# B&R Automation Studio project UdpReceiverSender
Automation Studio 4.5.3.86 SP

## Configuration Config1

CPU X20CP1585, AutomationRuntime A4.53, Build 4.1.2, Vc V4.52.0

### Task classes (Cpu.sw)
```
Cyclic#4:
  UDP <- UDP.prg
Libraries: AsUDP, runtime
```

### Hardware
```
X20CP1585 : X20CP1585 v1.6.0.0
  Connector IF2:
    ActivateDevice = 1
    Mode = Manual
    InternetAddress = 192.168.32.19
    SubnetMask = 255.255.255.0
  ConfigurationID = UdpReceiverSender_Config1
```

## Logical view

Binary libraries used (declarations not repeated): AsUDP

### Program Logical/UDP (ANSIC)

#### Udp.c - Init, cyclic, exit code
```c
#include <bur/plctypes.h>
#include <stdbool.h>

#ifdef _DEFAULT_INCLUDES
	#include <AsDefault.h>
#endif

void _INIT ProgramInit(void)
{
	UdpOpen_0.enable = true;
}

void _CYCLIC ProgramCyclic(void)
{
	//UdpOpen_0.pIfAddr = ;
	UdpOpen_0.port = 4711;
	//UdpOpen_0.options = ;
	UdpOpen(&UdpOpen_0);

	if(UdpOpen_0.status == ERR_OK)
		UdpOpen_0.enable = false;

	UdpRecv_0.enable = !UdpOpen_0.enable;
	UdpRecv_0.ident = UdpOpen_0.ident;
	UdpRecv_0.pData = (UDINT)&RecvBuffer[0];
	UdpRecv_0.datamax = sizeof(RecvBuffer);
	//UdpRecv_0.flags = ;
	UdpRecv_0.pIpAddr = (UDINT)&IpAddr;
	UdpRecv(&UdpRecv_0);

	if(UdpRecv_0.status == ERR_OK)
	{
		RecvCounter++;
		RecvLen = UdpRecv_0.recvlen;
		UdpSend_0.enable = true;
	}

	UdpSend_0.ident = UdpOpen_0.ident;
	UdpSend_0.pHost = (UDINT)&IpAddr;
	UdpSend_0.port = 4712;
	UdpSend_0.pData = (UDINT)&RecvBuffer[0];
	UdpSend_0.datalen = RecvLen;
	//UdpSend_0.flags = ;
	UdpSend(&UdpSend_0);

	if(UdpSend_0.status == ERR_OK)
		UdpSend_0.enable = false;
}

void _EXIT ProgramExit(void)
{
	do
	{
		UdpClose_0.enable = true;
		UdpClose_0.ident = UdpOpen_0.ident;
		UdpClose(&UdpClose_0);
	}while(UdpClose_0.status == ERR_FUB_BUSY);
}
```

#### Variables.var - Local variables
```iecst
VAR
	UdpClose_0 : UdpClose;
	UdpSend_0 : UdpSend;
	IpAddr : STRING[15];
	UdpOpen_0 : UdpOpen;
	UdpRecv_0 : UdpRecv;
	RecvBuffer : ARRAY[0..19] OF USINT;
	RecvCounter : USINT;
	RecvLen : UDINT;
END_VAR
```

Listed in the project but not available here: Logical/Global.typ, Logical/Global.var, Logical/Libraries, Logical/UDP/Types.typ
